FUNCTION_BLOCK EL2622
VAR
	{attribute addProperty Name "WcState"}
	_wcState : WcStateBase;
	{attribute addProperty Name "Info data"}
	_infoData : InfoDataBase;
	_io : EL2xx2_Data;
END_VAR

PROPERTY IO : REFERENCE TO EL2xx2_Data
GET
IO REF= _io;
END_GET
END_PROPERTY

PROPERTY WcState : REFERENCE TO WcStateBase
GET
WcState REF= _wcState;
END_GET
END_PROPERTY

END_FUNCTION_BLOCK

(* stored: Version 1.1.0.1, ProductVersion 3.1.4024.9
   POU EL2622: Id {715e3992-b02c-03dc-162f-c08af21b3524}, SpecialFunc None
   Property IO: Id {3cd4ce42-a1a8-01d5-1bb8-2c84b6ef3cf7}
   Get Get: Id {e717050e-d1ba-0e59-121c-8e444251a974}
   Property WcState: Id {baa0f524-5843-0d87-2830-31e7a465ee27}
   Get Get: Id {5e502170-7f95-06a5-3dde-dcbc13191322} *)
